FUNCTION_BLOCK PUBLIC FB_UR_PN_IO
VAR_IN_OUT
	Hardware : TYP_HW_UR_PN;
END_VAR
VAR_INPUT
END_VAR
VAR_OUTPUT
END_VAR
VAR
	_speedSlider : REAL;
END_VAR

// Future versions should include digital and analog IO too, wasn't necessary in this application

IF THIS^.Hardware.Out.O2TURIO[0].0 THEN // Speed slider mask to false when written
	IF _speedSlider = THIS^.SpeedSlider THEN
		THIS^.Hardware.Out.O2TURIO[0].0 := FALSE; 
	END_IF;
END_IF;

PROPERTY PUBLIC PumpVoltage : REAL
GET
VAR
	TempReal: REAL;
END_VAR
{warning disable C0371}

IF __ISVALIDREF(THIS^.Hardware) THEN

	FC_FLIP_DWORD(In := ADR(THIS^.Hardware.In.T2OURIO[16]), Out := ADR(TempReal));
	PumpVoltage := TempReal;
	
END_IF;
END_GET
END_PROPERTY

PROPERTY PUBLIC SpeedSlider : REAL
GET
VAR
	TempReal : REAL;
END_VAR
{warning disable C0371}

IF __ISVALIDREF(THIS^.Hardware) THEN

	FC_FLIP_DWORD(In := ADR(THIS^.Hardware.In.T2OURState[20]), Out := ADR(TempReal));
	SpeedSlider := TempReal;
	
END_IF;
END_GET
SET
{warning disable C0371}

IF __ISVALIDREF(THIS^.Hardware) THEN

	IF NOT THIS^.Hardware.Out.O2TURIO[0].0 THEN // Speed slider mask
		FC_FLIP_DWORD(In := ADR(SpeedSlider), Out := ADR(THIS^.Hardware.Out.O2TURIO[4]));
		_speedSlider := SpeedSlider;
		THIS^.Hardware.Out.O2TURIO[0].0 := TRUE; 
	END_IF
	
END_IF;
END_SET
END_PROPERTY

END_FUNCTION_BLOCK

(* stored: Version 1.1.0.1, ProductVersion 3.1.4024.12
   POU FB_UR_PN_IO: Id {539fe447-43b6-4c68-a860-e0e38ba41bc7}, SpecialFunc None
   Property PumpVoltage: Id {31b5347a-947f-49eb-8112-982d3689c3ba}
   Get Get: Id {6896f5b8-1d0c-422b-aea8-77e7fcb0db3c}
   Property SpeedSlider: Id {283e5a7f-0140-4689-8d08-35fe883aa469}
   Get Get: Id {40d964fa-1e9f-426e-88dd-8a7d1b03f4e5}
   Set Set: Id {49f6c1d4-970e-44b6-b56a-36d7631cc0fd} *)
